% RSLogix 500 project Job 14 - Leo Kniffen.RSS, saved by version 10.00.00.00 %
PROJECT "ML04B"    % processor: Bul.1763 MicroLogix 1100 Series B %

PROGRAM FILES
  LAD 2   10 rungs

DATA FILES
  O0 OUTPUT  4 elements
  I1 INPUT  6 elements
  S2 STATUS  66 elements
  B3 BINARY  1 elements
  T4 TIMER  1 elements
  C5 COUNTER  1 elements
  R6 CONTROL  1 elements
  N7 INTEGER  1 elements
  F8 FLOAT  1 elements

LADDER 2
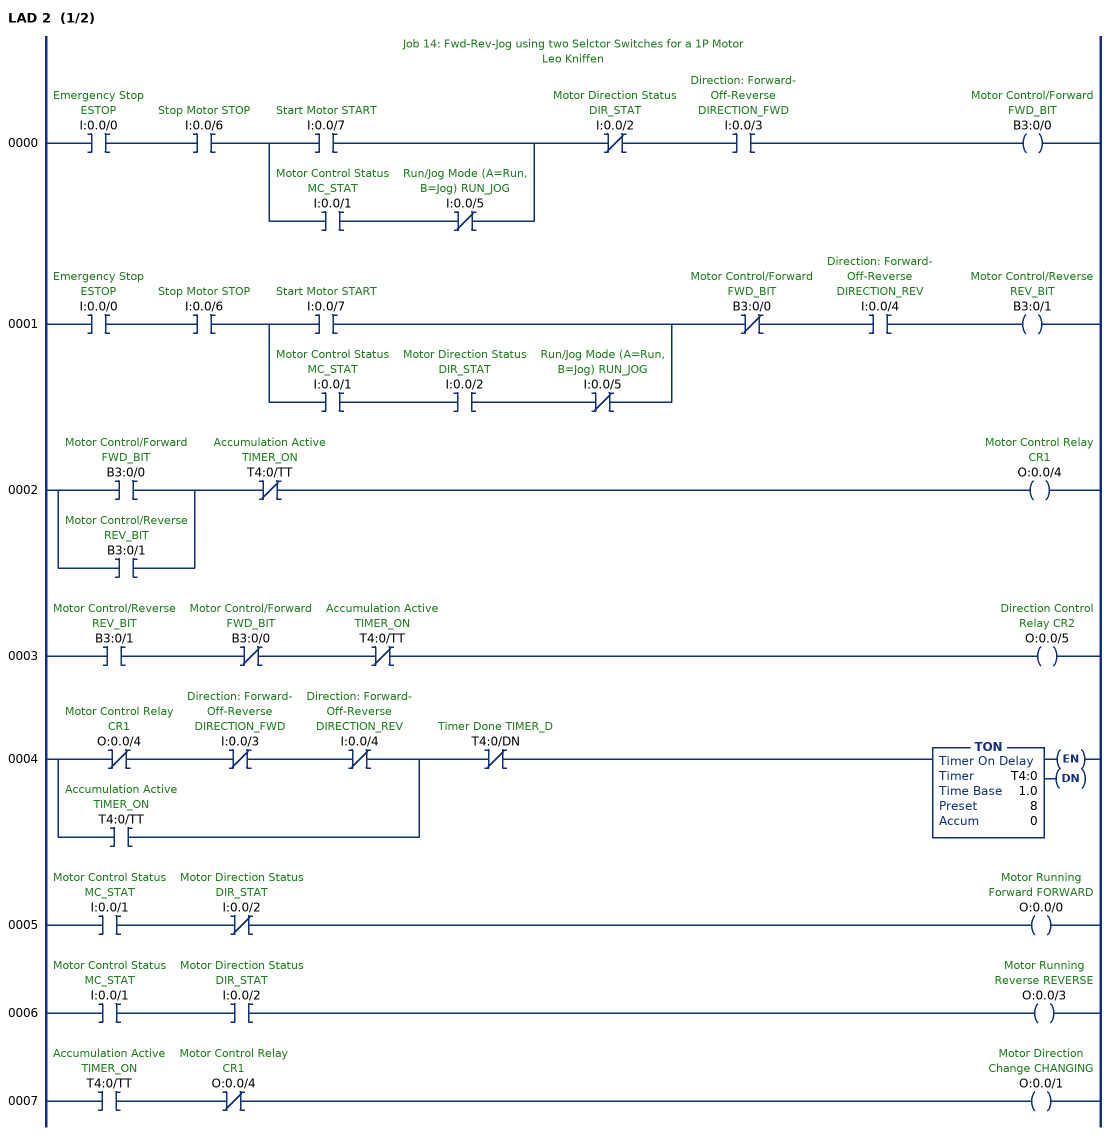
% Rung: 0 %
% Job 14: Fwd-Rev-Jog using two Selctor Switches for a 1P Motor
% Leo Kniffen %
SOR XIC I:0.0/0 XIC I:0.0/6 BST XIC I:0.0/7 NXB XIC I:0.0/1 XIO I:0.0/5 BND XIO I:0.0/2 XIC I:0.0/3 OTE B3:0/0 EOR
%   I:0.0/0  ESTOP  "Emergency Stop" %
%   I:0.0/6  STOP  "Stop Motor" %
%   I:0.0/7  START  "Start Motor" %
%   I:0.0/1  MC_STAT  "Motor Control Status" %
%   I:0.0/5  RUN_JOG  "Run/Jog Mode (A=Run, B=Jog)" %
%   I:0.0/2  DIR_STAT  "Motor Direction Status" %
%   I:0.0/3  DIRECTION_FWD  "Direction: Forward- Off-Reverse" %
%   B3:0/0  FWD_BIT  "Motor Control/Forward" %
% Rung: 1 %
SOR XIC I:0.0/0 XIC I:0.0/6 BST XIC I:0.0/7 NXB XIC I:0.0/1 XIC I:0.0/2 XIO I:0.0/5 BND XIO B3:0/0 XIC I:0.0/4 OTE B3:0/1 EOR
%   I:0.0/0  ESTOP  "Emergency Stop" %
%   I:0.0/6  STOP  "Stop Motor" %
%   I:0.0/7  START  "Start Motor" %
%   I:0.0/1  MC_STAT  "Motor Control Status" %
%   I:0.0/2  DIR_STAT  "Motor Direction Status" %
%   I:0.0/5  RUN_JOG  "Run/Jog Mode (A=Run, B=Jog)" %
%   B3:0/0  FWD_BIT  "Motor Control/Forward" %
%   I:0.0/4  DIRECTION_REV  "Direction: Forward- Off-Reverse" %
%   B3:0/1  REV_BIT  "Motor Control/Reverse" %
% Rung: 2 %
SOR BST XIC B3:0/0 NXB XIC B3:0/1 BND XIO T4:0/TT OTE O:0.0/4 EOR
%   B3:0/0  FWD_BIT  "Motor Control/Forward" %
%   B3:0/1  REV_BIT  "Motor Control/Reverse" %
%   T4:0/TT  TIMER_ON  "Accumulation Active" %
%   O:0.0/4  CR1  "Motor Control Relay" %
% Rung: 3 %
SOR XIC B3:0/1 XIO B3:0/0 XIO T4:0/TT OTE O:0.0/5 EOR
%   B3:0/1  REV_BIT  "Motor Control/Reverse" %
%   B3:0/0  FWD_BIT  "Motor Control/Forward" %
%   T4:0/TT  TIMER_ON  "Accumulation Active" %
%   O:0.0/5  CR2  "Direction Control Relay" %
% Rung: 4 %
SOR BST XIO O:0.0/4 XIO I:0.0/3 XIO I:0.0/4 NXB XIC T4:0/TT BND XIO T4:0/DN TON T4:0 1.0 8 0 EOR
%   O:0.0/4  CR1  "Motor Control Relay" %
%   I:0.0/3  DIRECTION_FWD  "Direction: Forward- Off-Reverse" %
%   I:0.0/4  DIRECTION_REV  "Direction: Forward- Off-Reverse" %
%   T4:0/TT  TIMER_ON  "Accumulation Active" %
%   T4:0/DN  TIMER_D  "Timer Done" %
% Rung: 5 %
SOR XIC I:0.0/1 XIO I:0.0/2 OTE O:0.0/0 EOR
%   I:0.0/1  MC_STAT  "Motor Control Status" %
%   I:0.0/2  DIR_STAT  "Motor Direction Status" %
%   O:0.0/0  FORWARD  "Motor Running Forward" %
% Rung: 6 %
SOR XIC I:0.0/1 XIC I:0.0/2 OTE O:0.0/3 EOR
%   I:0.0/1  MC_STAT  "Motor Control Status" %
%   I:0.0/2  DIR_STAT  "Motor Direction Status" %
%   O:0.0/3  REVERSE  "Motor Running Reverse" %
% Rung: 7 %
SOR XIC T4:0/TT XIO O:0.0/4 OTE O:0.0/1 EOR
%   T4:0/TT  TIMER_ON  "Accumulation Active" %
%   O:0.0/4  CR1  "Motor Control Relay" %
%   O:0.0/1  CHANGING  "Motor Direction Change" %

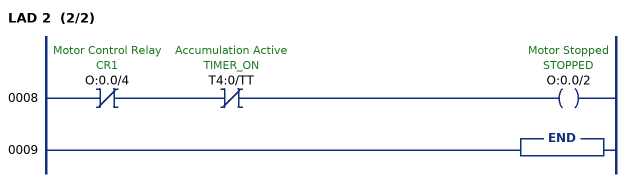
% Rung: 8 %
SOR XIO O:0.0/4 XIO T4:0/TT OTE O:0.0/2 EOR
%   O:0.0/4  CR1  "Motor Control Relay" %
%   T4:0/TT  TIMER_ON  "Accumulation Active" %
%   O:0.0/2  STOPPED  "Motor Stopped" %
% Rung: 9 %
SOR END EOR

OTHER DOCUMENTED ADDRESSES
  B3:0/2  FWD_SAVED  "Saved forward bit"
  B3:0/3  REV_SAVED  "Saved reverse bit"
  I:0.0/8  REV  "Motor Reverse"
  T4:0/EN  TIMER_E  "Timer enable"

DATA TABLE (non-zero values as saved)
DATA T4
% .PRE .ACC %
% T4:0 % 8 0
